Staubli VAL3: onBackEvent.pgx

program onBackEvent(string x_sId, bool& x_bSave[])
  local bool l_bFound
  local num l_nX
  local num l_nY
  local string l_sString
  local string l_sMessage
  local bool l_bOk
  local num l_nValue
begin
  //
  // NB sEvent is the selected
  // element in the LIST
  //
  switch nViewMode
    case 0,1
      // OUT IN NUM
      call onEnterEvent(x_sId,x_bSave)
    break
    case 2
      // COUNT
      l_nX=40-use:nBottomX+find(sEvent,"{")
      call saveInOut:getItem_num(l_sString,x_sId)
      l_nY=nView+1
      // clean the line
      call use:listcursor(use:nView,false)
      // read the name
      call use:read(l_nX,l_nY,l_sString,14,false)
      // check if already exist
      if !use:bUseEscape and l_sString!=""
        // set the value
        call NUM:set(l_sString,x_sId)
      endIf
      // save it
      x_bSave=true
    break
  endSwitch
end
